(* PLC project Unnamed, Unknown Unnamed 1 *)
(* stored: creationDateTime 2023-03-10T10:37:17, modificationDateTime 2023-03-15T15:56:42 *)

(* https://www.gds2.de/fileadmin/umwelttechnik/umwelttechnik/skripte/steuerungstechnik_ut_2017.pdf, 2.11 *)
FUNCTION_BLOCK Pollutant_Indicator
  VAR_INPUT
    IN1 : BOOL;
    IN2 : BOOL;
    IN3 : BOOL;
  END_VAR
  VAR_OUTPUT
    OUT1 : BOOL;
    OUT2 : BOOL;
    OUT3 : BOOL;
  END_VAR

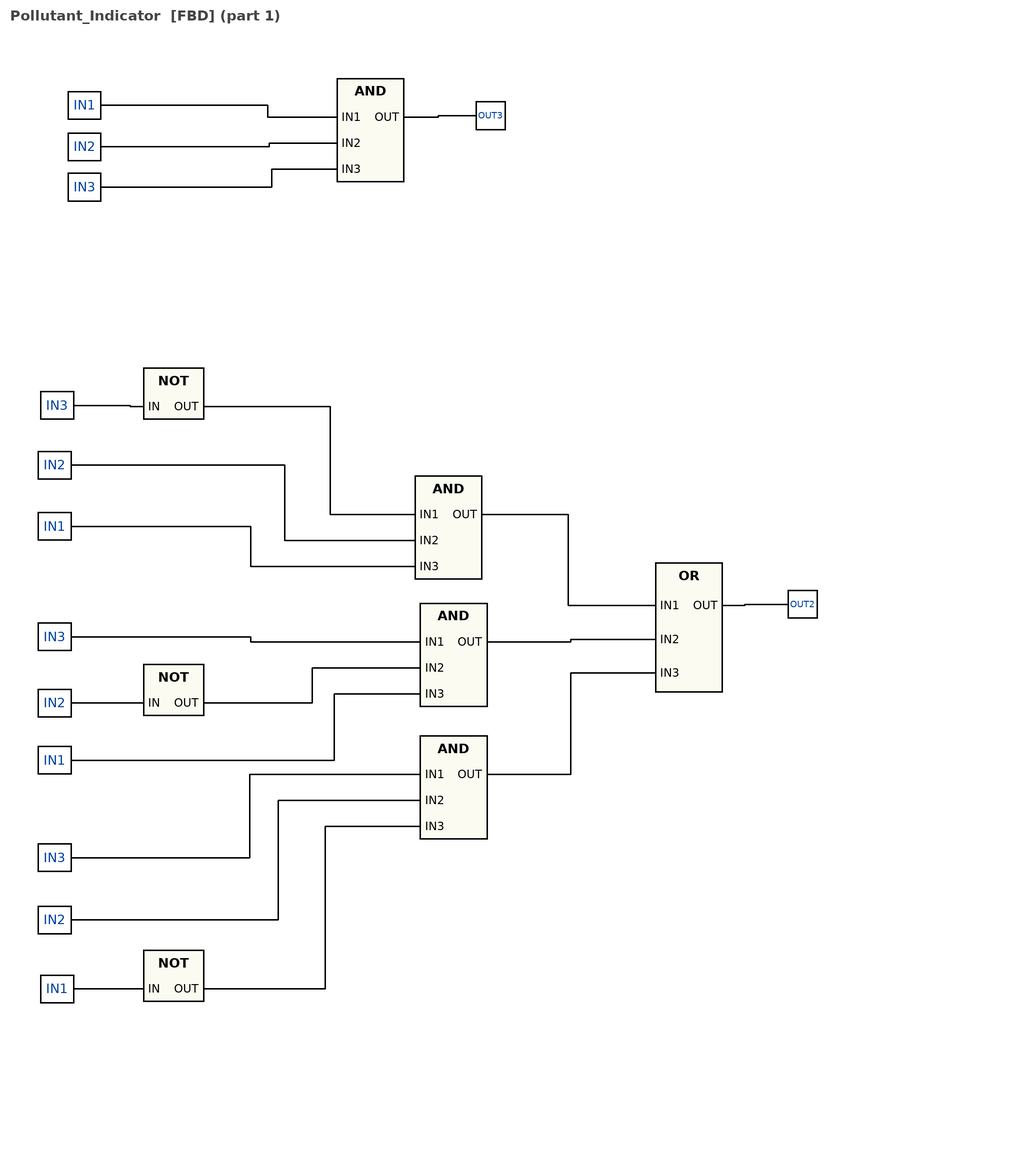
(* FBD diagram, written out as Structured Text *)
OUT3 := IN1 AND IN2 AND IN3;
OUT2 := NOT IN3 AND IN2 AND IN1 OR IN3 AND NOT IN2 AND IN1 OR IN3 AND IN2 AND NOT IN1;
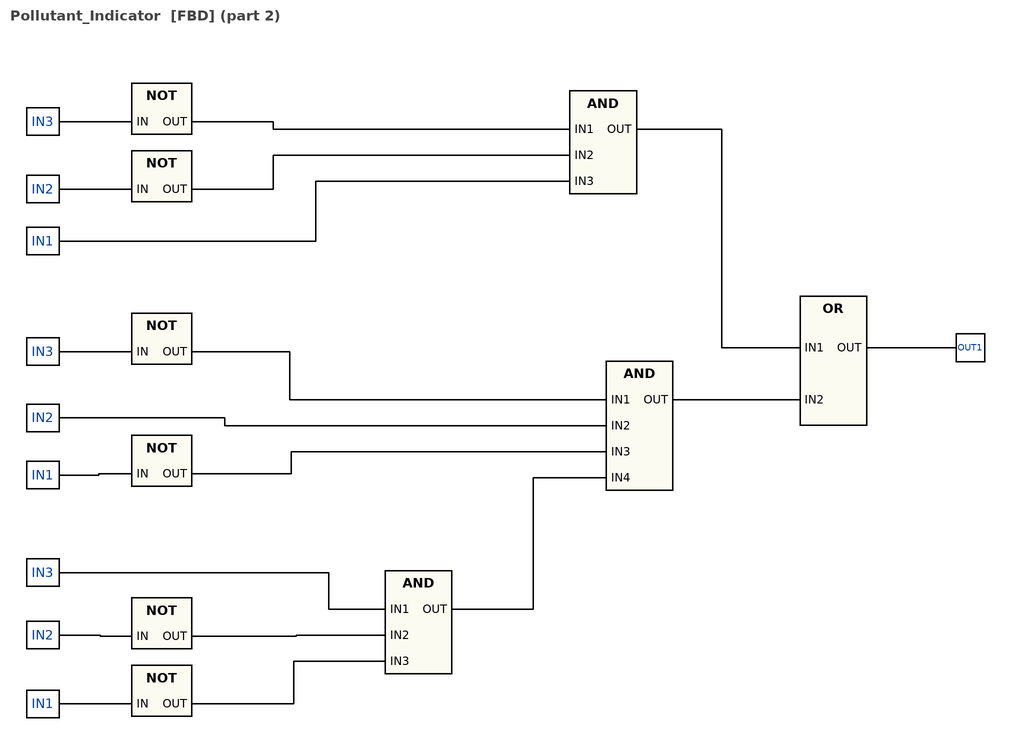
OUT1 := NOT IN3 AND NOT IN2 AND IN1 OR NOT IN3 AND IN2 AND NOT IN1 AND IN3 AND NOT IN2 AND NOT IN1;
END_FUNCTION_BLOCK

CONFIGURATION config
  RESOURCE resource1 ON PLC
  END_RESOURCE
END_CONFIGURATION
